(* PLC project Unnamed, 不明 Unnamed 1 *)
(* stored: creationDateTime 2021-07-12T09:24:00, modificationDateTime 2021-08-19T15:03:51 *)

PROGRAM va_control
  VAR
    Va_AD AT %IW102 : WORD;  (* A/D変換 Va *)
    Nm_AD AT %IW103 : WORD;  (* A/D変換 Nm *)
  END_VAR
  VAR
    Vref : REAL := 0.0;  (* Va* REAL演算用 *)
    Va : REAL := 0.0;  (* Va REAL演算用 *)
    Duty_Va : REAL := 0.0;
  END_VAR
  VAR
    PWM1 AT %QW101 : WORD;  (* Va制御用 *)
  END_VAR
  VAR
    R_run : BOOL;  (* 実験実行フラグ *)
  END_VAR
  VAR
    R1 AT %QX100.2 : BOOL;  (* 電源 %QX100.2 *)
    R2 AT %QX100.3 : BOOL;  (* 電源 %QX100.3 *)
  END_VAR
  VAR
    Rtim0 : BOOL;
    Rtim1 : BOOL;
    Rtim2 : BOOL;
    Rtim3 : BOOL;
    Rtim4 : BOOL;
  END_VAR
  VAR
    Run AT %IX100.0 : BOOL;  (* 実験開始ボタン *)
    Stop AT %IX100.1 : BOOL;  (* 実験停止ボタン *)
    G_reset AT %QX100.1 : BOOL;  (* ゲートリセット *)
  END_VAR
  VAR
    TON1 : TON;
    TON0 : TON;
    RAMP0 : RAMP;
    TON2 : TON;
    TON3 : TON;
    TON4 : TON;
    TON5 : TON;
    RAMP1 : RAMP;
    RAMP2 : RAMP;
    RAMP3 : RAMP;
    RAMP5 : RAMP;
    INTEGRAL0 : INTEGRAL;
    TON6 : TON;
  END_VAR
  VAR  (* added by the conversion: wires and edge detectors of the diagram *)
    _SUB216_ENO : BOOL;
    _SUB216_OUT : REAL;
    _MUL219_ENO : BOOL;
    _MUL219_OUT : REAL;
    _ADD224_OUT : ANY;
    _LIMIT225_OUT : ANY;
    _MUL233_ENO : BOOL;
    _MUL233_OUT : REAL;
    _ADD224_ENO : BOOL;
    _LIMIT225_ENO : BOOL;
  END_VAR

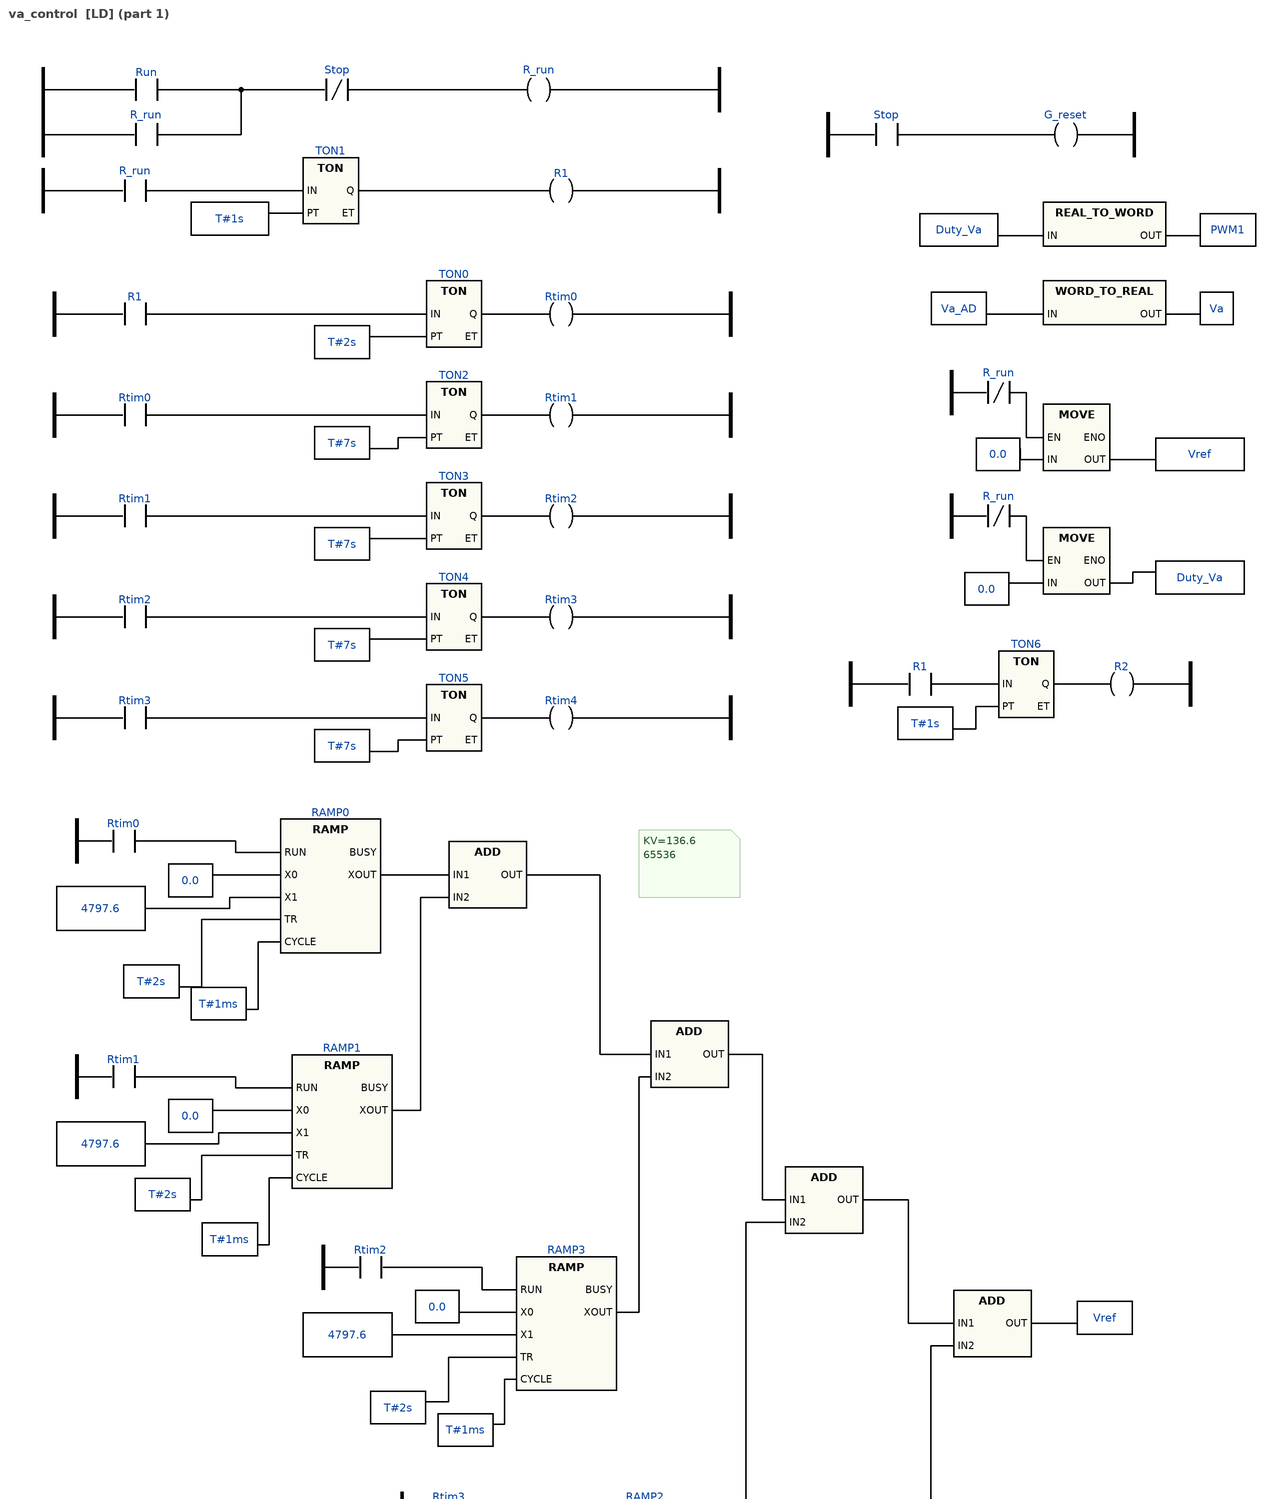
(* LD diagram, written out as Structured Text *)
R_run := (Run OR R_run) AND NOT Stop;
G_reset := Stop;
TON1(IN := R_run, PT := T#1s);
R1 := TON1.Q;
PWM1 := REAL_TO_WORD(Duty_Va);
Va := WORD_TO_REAL(Va_AD);
TON0(IN := R1, PT := T#2s);
Rtim0 := TON0.Q;
TON2(IN := Rtim0, PT := T#7s);
Rtim1 := TON2.Q;
IF NOT R_run THEN Vref := 0.0; END_IF;
TON3(IN := Rtim1, PT := T#7s);
Rtim2 := TON3.Q;
IF NOT R_run THEN Duty_Va := 0.0; END_IF;
TON4(IN := Rtim2, PT := T#7s);
Rtim3 := TON4.Q;
TON6(IN := R1, PT := T#1s);
R2 := TON6.Q;
TON5(IN := Rtim3, PT := T#7s);
Rtim4 := TON5.Q;
(* KV=136.6
65536 *)
RAMP0(RUN := Rtim0, X0 := 0.0, X1 := 4797.6, TR := T#2s, CYCLE := T#1ms);
RAMP1(RUN := Rtim1, X0 := 0.0, X1 := 4797.6, TR := T#2s, CYCLE := T#1ms);
RAMP3(RUN := Rtim2, X0 := 0.0, X1 := 4797.6, TR := T#2s, CYCLE := T#1ms);
RAMP2(RUN := Rtim3, X0 := 0.0, X1 := 4797.6, TR := T#2s, CYCLE := T#1ms);
RAMP5(RUN := Rtim4, X0 := 0.0, X1 := 4797.6, TR := T#2s, CYCLE := T#1ms);
Vref := RAMP0.XOUT + RAMP1.XOUT + RAMP3.XOUT + RAMP2.XOUT + RAMP5.XOUT;
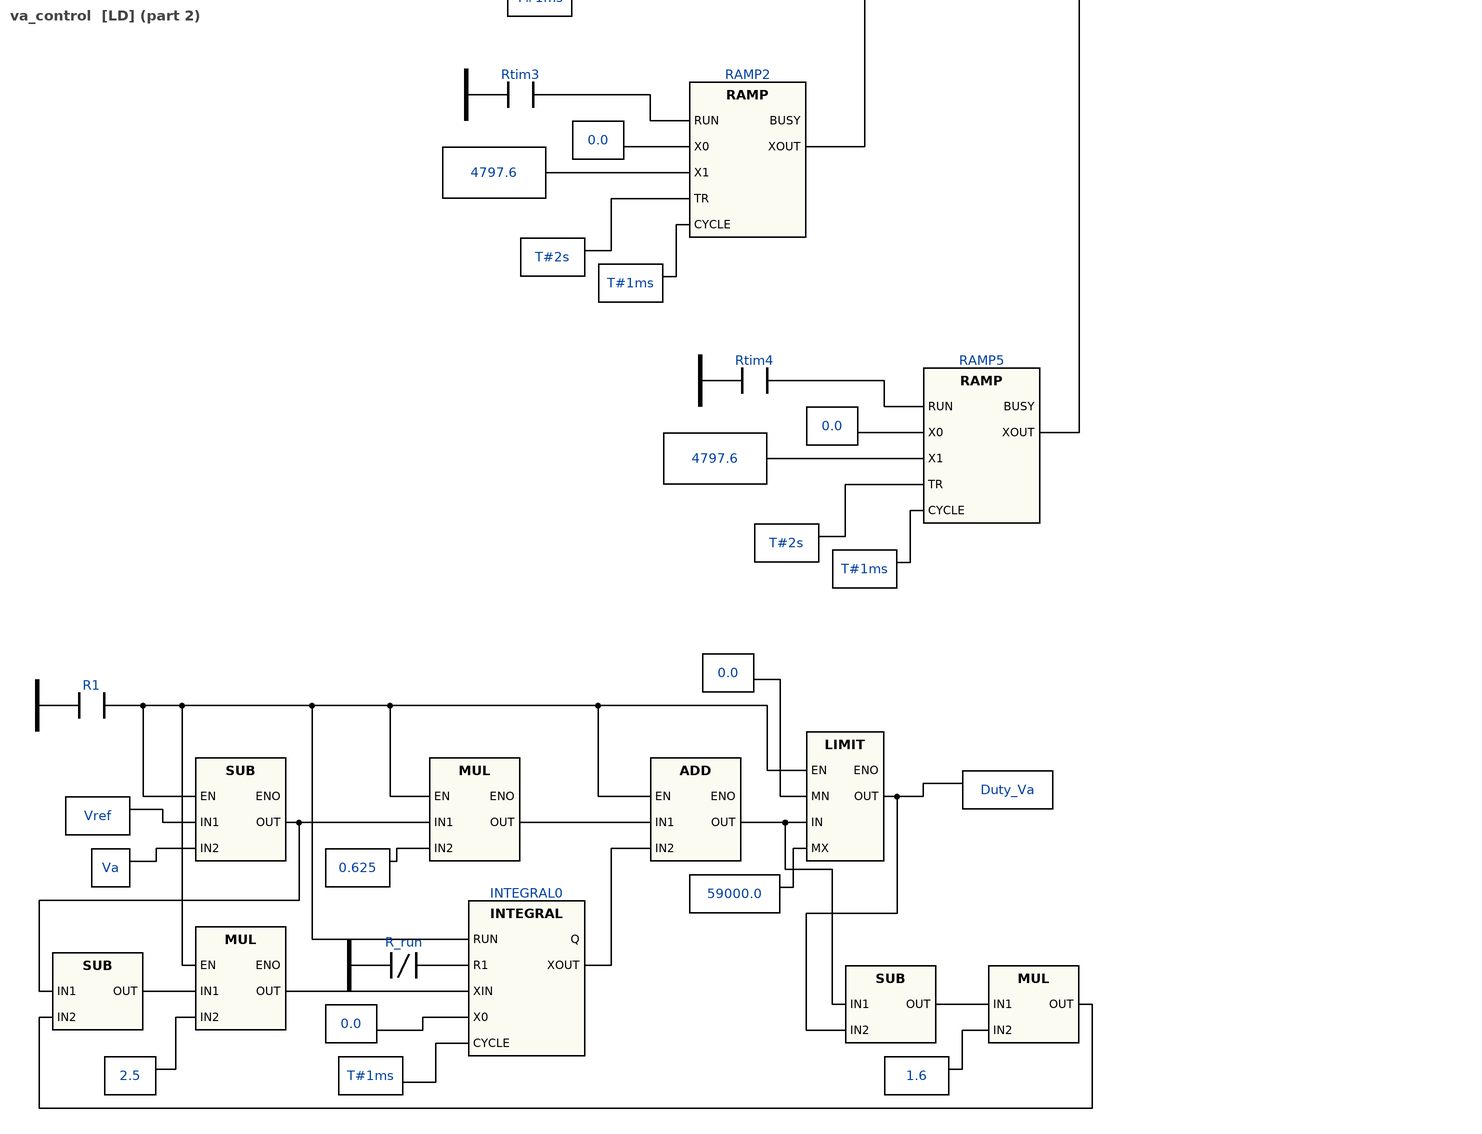
_SUB216_OUT := SUB(EN := R1, IN1 := Vref, IN2 := Va, ENO => _SUB216_ENO);
_MUL219_OUT := MUL(EN := R1, IN1 := _SUB216_OUT, IN2 := 0.625, ENO => _MUL219_ENO);
_MUL233_OUT := MUL(EN := R1, IN1 := _SUB216_OUT - (_ADD224_OUT - _LIMIT225_OUT) * 1.6, IN2 := 2.5, ENO => _MUL233_ENO);
INTEGRAL0(RUN := R1, R1 := NOT R_run, XIN := _MUL233_OUT, X0 := 0.0, CYCLE := T#1ms);
_ADD224_OUT := ADD(EN := R1, IN1 := _MUL219_OUT, IN2 := INTEGRAL0.XOUT, ENO => _ADD224_ENO);
_LIMIT225_OUT := LIMIT(EN := R1, MN := 0.0, IN := _ADD224_OUT, MX := 59000.0, ENO => _LIMIT225_ENO);
IF _LIMIT225_ENO THEN Duty_Va := _LIMIT225_OUT; END_IF;
END_PROGRAM

CONFIGURATION Config0
  RESOURCE Res0 ON PLC
    TASK task0(INTERVAL := T#1ms, PRIORITY := 0);
    PROGRAM instance0 WITH task0 : va_control;
  END_RESOURCE
END_CONFIGURATION
